Omron CX-Programmer project 新工程 (CX-Programmer 9.72)

# PLC 新PLC1: CP1E E40

## Global symbols (name address type ; comment)
0.00 BOOL  ; 回程1
0.01 BOOL  ; 刹车信号1
0.02 BOOL  ; 系统正常
0.03 BOOL  ; 超程
0.04 BOOL  ; 吹件
0.05 BOOL  ; 刹车信号子2
0.06 BOOL  ; 光电控制1
0.07 BOOL  ; 计数值到
0.08 BOOL  ; 电机启动
0.09 BOOL  ; 电机停止
0.10 BOOL  ; 电机正转
0.11 BOOL  ; 电机反转
100.01 BOOL  ; 运转侦查1
100.02 BOOL  ; 超程指示
100.03 BOOL  ; 凸轮故障
100.04 BOOL  ; 吹件阀
100.05 BOOL  ; 气动泵控制阀
100.06 BOOL  ; 吹件阀2
100.07 BOOL  ; 油泵电机
101.00 BOOL  ; 电机正转
101.01 BOOL  ; 电机反转
101.02 BOOL  ; △运行
101.03 BOOL  ; Y启动
101.04 BOOL  ; 气压指示
101.05 BOOL  ; 连续预置
101.07 BOOL  ; 电机运行
102.00 BOOL  ; 运行侦测2
102.01 BOOL  ; 顶点补正
102.02 BOOL  ; 保护继电器
102.03 BOOL  ; 辅助调整2
102.04 BOOL  ; 润滑故障
102.05 BOOL  ; 双联阀故障指示
102.06 BOOL  ; 异常报警
102.07 BOOL  ; 负荷指示
10.01 BOOL  ; 自动送料阀
13.01 BOOL  ; 电机正反转信号
13.04 BOOL  ; 电机启动信号
14.03 BOOL  ; 运行条件
14.04 BOOL  ; 寸动规范输出
14.05 BOOL  ; 双手同步输出信号
14.06 BOOL  ; 单次信号输出
14.07 BOOL  ; 连续预置信号
14.08 BOOL  ; 误送信号
15.00 BOOL  ; 寸动输出
15.01 BOOL  ; 单次输出
15.03 BOOL  ; 连续输出
15.04 BOOL  ; 调整规范
15.05 BOOL  ; 脚踏输出信号
16.00 BOOL  ; 1秒故障闪烁信号
16.01 BOOL  ; 故障输出
17.00 BOOL  ; 寸动光电遮断信号
18.01 BOOL  ; 功能开关拨动信号
18.03 BOOL  ; 双联阀故障
19.01 BOOL  ; 连续停止信号
19.02 BOOL  ; 连续信号输出
19.05 BOOL  ; 单次运行条件
1.00 BOOL  ; 光电保护
1.01 BOOL  ; 超负荷
1.02 BOOL  ; 脚踏旋钮
1.03 BOOL  ; 双手A
1.04 BOOL  ; 双手B
1.05 BOOL  ; 连续预置
1.06 BOOL  ; 连续停止
1.07 BOOL  ; 急停
1.08 BOOL  ; 气压
1.09 BOOL  ; 送料许可
1.10 BOOL  ; 双联阀故障检测
1.11 BOOL  ; 脚踏开关
200.00 BOOL  ; 润滑屏蔽
200.01 BOOL  ; 气压传感屏蔽
20.02 BOOL  ; 双联阀下降沿
20.03 BOOL  ; 二度落动作
20.04 BOOL  ; 二度落保护
20.05 BOOL  ; 上死点停车
20.06 BOOL  ; 二度落保护
20.07 BOOL  ; 超程保护
22.00 BOOL  ; 单次回程前信号
22.01 BOOL  ; 回程后断回程前
23.00 BOOL  ; 连续信号开始
24.02 BOOL  ; 调整
24.03 BOOL  ; 连续顶点补正信号
24.05 BOOL  ; 反馈不同步
29.00 BOOL  ; 二度落上升沿
29.02 BOOL  ; 超程下降沿
2.00 BOOL  ; 反馈信号1
2.01 BOOL  ; 异常复位
2.02 BOOL  ; 润滑故障检测
2.03 BOOL  ; 寸动信号
2.04 BOOL  ; 单次信号
2.05 BOOL  ; 连续信号
2.06 BOOL  ; 送料接口
2.07 BOOL  ; 误送检知
2.08 BOOL  ; 光电控制2
2.10 BOOL  ; 自动送料
2.11 BOOL  ; 二度落
30.08 BOOL  ; 润滑故障信号
T004 BOOL  ; 双手同步时间
T006 BOOL  ; 连续预置时间
T007 BOOL  ; Y-三角转换时间
T009 BOOL  ; 超负荷信号
T015 BOOL  ; 二度落异常
T018 BOOL  ; 润滑检测开关常通
T019 BOOL  ; 润滑检测开关常闭
T040 BOOL  ; 急停滤波
T042 BOOL  ; 单次双手时间
T045 BOOL  ; 压力处理信号

## Program 新程序1 (cyclic task 0)
Local symbols
p_on BOOL
y20 BOOL

### Section 段1

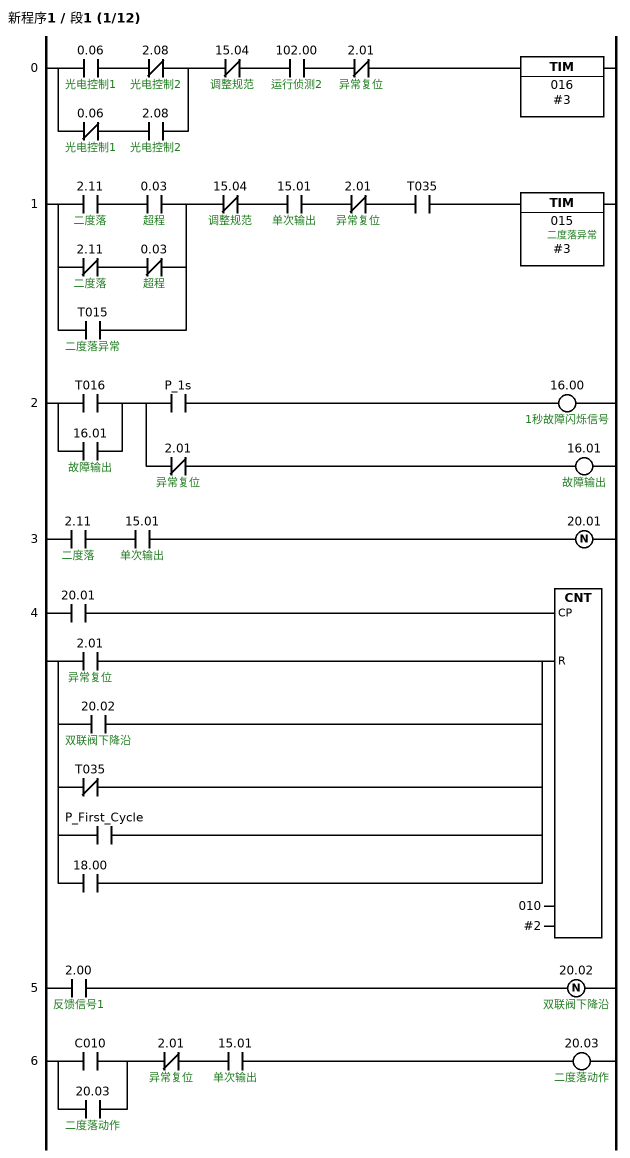
; rung 0
LD 0.06  ; 光电控制1
ANDNOT 2.08  ; 光电控制2
LDNOT 0.06  ; 光电控制1
AND 2.08  ; 光电控制2
ORLD
ANDNOT 15.04  ; 调整规范
AND 102.00  ; 运行侦测2
ANDNOT 2.01  ; 异常复位
TIM 016 #3
; rung 1
LD 2.11  ; 二度落
AND 0.03  ; 超程
LDNOT 2.11  ; 二度落
ANDNOT 0.03  ; 超程
ORLD
OR T015  ; 二度落异常
ANDNOT 15.04  ; 调整规范
AND 15.01  ; 单次输出
ANDNOT 2.01  ; 异常复位
AND T035
TIM 015 #3  ; 二度落异常
; rung 2
LD T016
OR 16.01  ; 故障输出
OUT TR0
AND P_1s
OUT 16.00  ; 1秒故障闪烁信号
LD TR0
ANDNOT 2.01  ; 异常复位
OUT 16.01  ; 故障输出
; rung 3
LD 2.11  ; 二度落
AND 15.01  ; 单次输出
DIFD(014) 20.01
; rung 4
LD 20.01
LD 2.01  ; 异常复位
OR 20.02  ; 双联阀下降沿
ORNOT T035
OR P_First_Cycle
OR 18.00
CNT 010 #2
; rung 5
LD 2.00  ; 反馈信号1
DIFD(014) 20.02  ; 双联阀下降沿
; rung 6
LD C010
OR 20.03  ; 二度落动作
ANDNOT 2.01  ; 异常复位
AND 15.01  ; 单次输出
OUT 20.03  ; 二度落动作

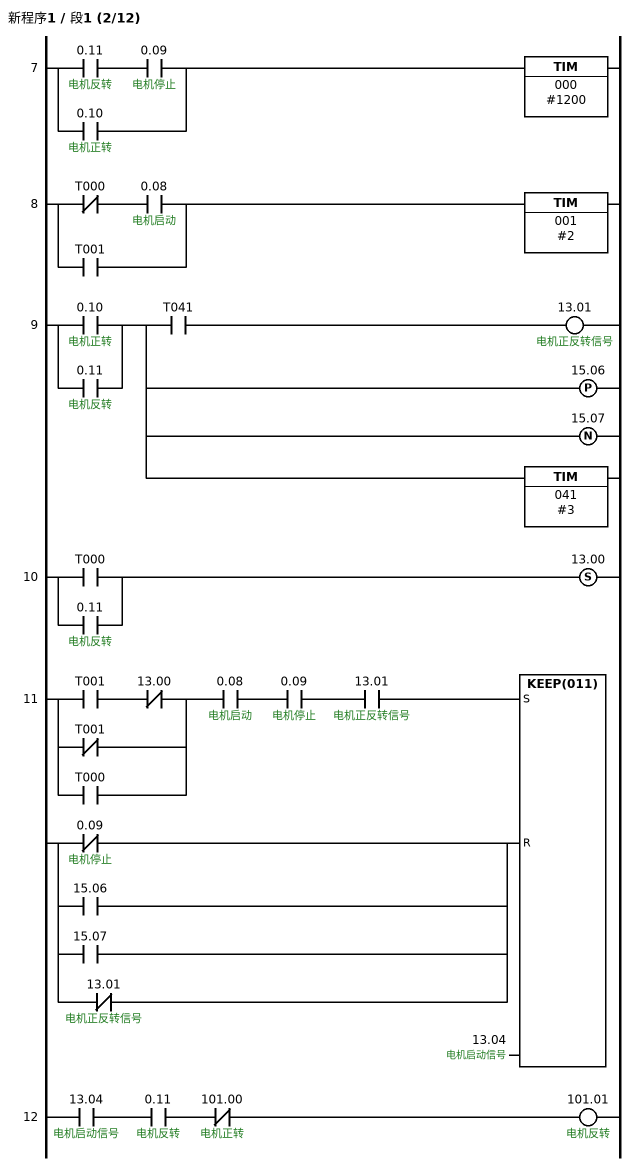
; rung 7
LD 0.11  ; 电机反转
AND 0.09  ; 电机停止
OR 0.10  ; 电机正转
TIM 000 #1200
; rung 8
LDNOT T000
AND 0.08  ; 电机启动
OR T001
TIM 001 #2
; rung 9
LD 0.10  ; 电机正转
OR 0.11  ; 电机反转
OUT TR0
AND T041
OUT 13.01  ; 电机正反转信号
LD TR0
DIFU(013) 15.06
DIFD(014) 15.07
TIM 041 #3
; rung 10
LD T000
OR 0.11  ; 电机反转
SET 13.00
; rung 11
LD T001
ANDNOT 13.00
ORNOT T001
OR T000
AND 0.08  ; 电机启动
AND 0.09  ; 电机停止
AND 13.01  ; 电机正反转信号
LDNOT 0.09  ; 电机停止
OR 15.06
OR 15.07
ORNOT 13.01  ; 电机正反转信号
KEEP(011) 13.04  ; 电机启动信号
; rung 12
LD 13.04  ; 电机启动信号
AND 0.11  ; 电机反转
ANDNOT 101.00  ; 电机正转
OUT 101.01  ; 电机反转

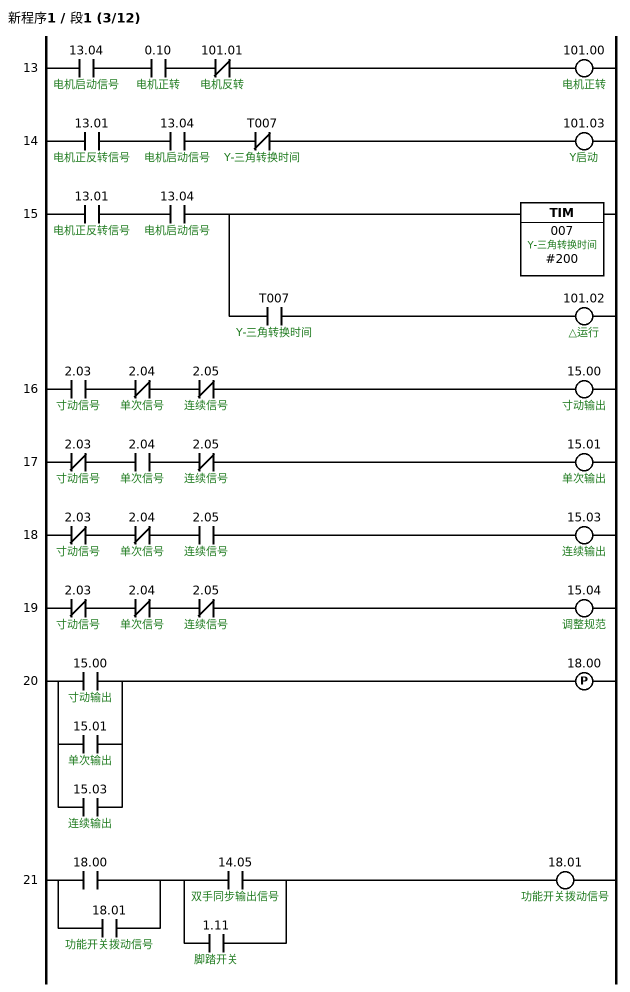
; rung 13
LD 13.04  ; 电机启动信号
AND 0.10  ; 电机正转
ANDNOT 101.01  ; 电机反转
OUT 101.00  ; 电机正转
; rung 14
LD 13.01  ; 电机正反转信号
AND 13.04  ; 电机启动信号
ANDNOT T007  ; Y-三角转换时间
OUT 101.03  ; Y启动
; rung 15
LD 13.01  ; 电机正反转信号
AND 13.04  ; 电机启动信号
TIM 007 #200  ; Y-三角转换时间
AND T007  ; Y-三角转换时间
OUT 101.02  ; △运行
; rung 16
LD 2.03  ; 寸动信号
ANDNOT 2.04  ; 单次信号
ANDNOT 2.05  ; 连续信号
OUT 15.00  ; 寸动输出
; rung 17
LDNOT 2.03  ; 寸动信号
AND 2.04  ; 单次信号
ANDNOT 2.05  ; 连续信号
OUT 15.01  ; 单次输出
; rung 18
LDNOT 2.03  ; 寸动信号
ANDNOT 2.04  ; 单次信号
AND 2.05  ; 连续信号
OUT 15.03  ; 连续输出
; rung 19
LDNOT 2.03  ; 寸动信号
ANDNOT 2.04  ; 单次信号
ANDNOT 2.05  ; 连续信号
OUT 15.04  ; 调整规范
; rung 20
LD 15.00  ; 寸动输出
OR 15.01  ; 单次输出
OR 15.03  ; 连续输出
DIFU(013) 18.00
; rung 21
LD 18.00
OR 18.01  ; 功能开关拨动信号
LD 14.05  ; 双手同步输出信号
OR 1.11  ; 脚踏开关
ANDLD
OUT 18.01  ; 功能开关拨动信号

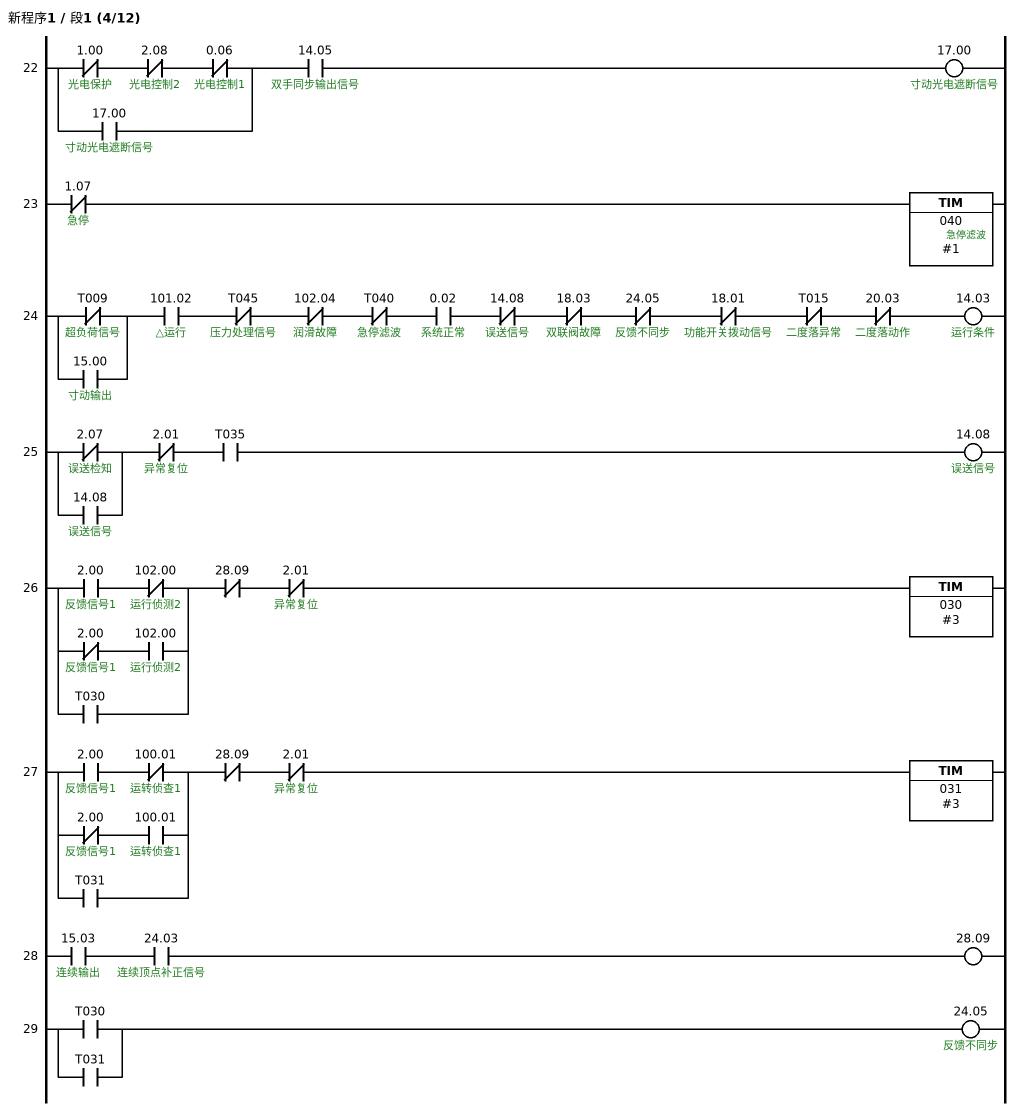
; rung 22
LDNOT 1.00  ; 光电保护
ANDNOT 2.08  ; 光电控制2
ANDNOT 0.06  ; 光电控制1
OR 17.00  ; 寸动光电遮断信号
AND 14.05  ; 双手同步输出信号
OUT 17.00  ; 寸动光电遮断信号
; rung 23
LDNOT 1.07  ; 急停
TIM 040 #1  ; 急停滤波
; rung 24
LDNOT T009  ; 超负荷信号
OR 15.00  ; 寸动输出
AND 101.02  ; △运行
ANDNOT T045  ; 压力处理信号
ANDNOT 102.04  ; 润滑故障
ANDNOT T040  ; 急停滤波
AND 0.02  ; 系统正常
ANDNOT 14.08  ; 误送信号
ANDNOT 18.03  ; 双联阀故障
ANDNOT 24.05  ; 反馈不同步
ANDNOT 18.01  ; 功能开关拨动信号
ANDNOT T015  ; 二度落异常
ANDNOT 20.03  ; 二度落动作
OUT 14.03  ; 运行条件
; rung 25
LDNOT 2.07  ; 误送检知
OR 14.08  ; 误送信号
ANDNOT 2.01  ; 异常复位
AND T035
OUT 14.08  ; 误送信号
; rung 26
LD 2.00  ; 反馈信号1
ANDNOT 102.00  ; 运行侦测2
LDNOT 2.00  ; 反馈信号1
AND 102.00  ; 运行侦测2
ORLD
OR T030
ANDNOT 28.09
ANDNOT 2.01  ; 异常复位
TIM 030 #3
; rung 27
LD 2.00  ; 反馈信号1
ANDNOT 100.01  ; 运转侦查1
LDNOT 2.00  ; 反馈信号1
AND 100.01  ; 运转侦查1
ORLD
OR T031
ANDNOT 28.09
ANDNOT 2.01  ; 异常复位
TIM 031 #3
; rung 28
LD 15.03  ; 连续输出
AND 24.03  ; 连续顶点补正信号
OUT 28.09
; rung 29
LD T030
OR T031
OUT 24.05  ; 反馈不同步

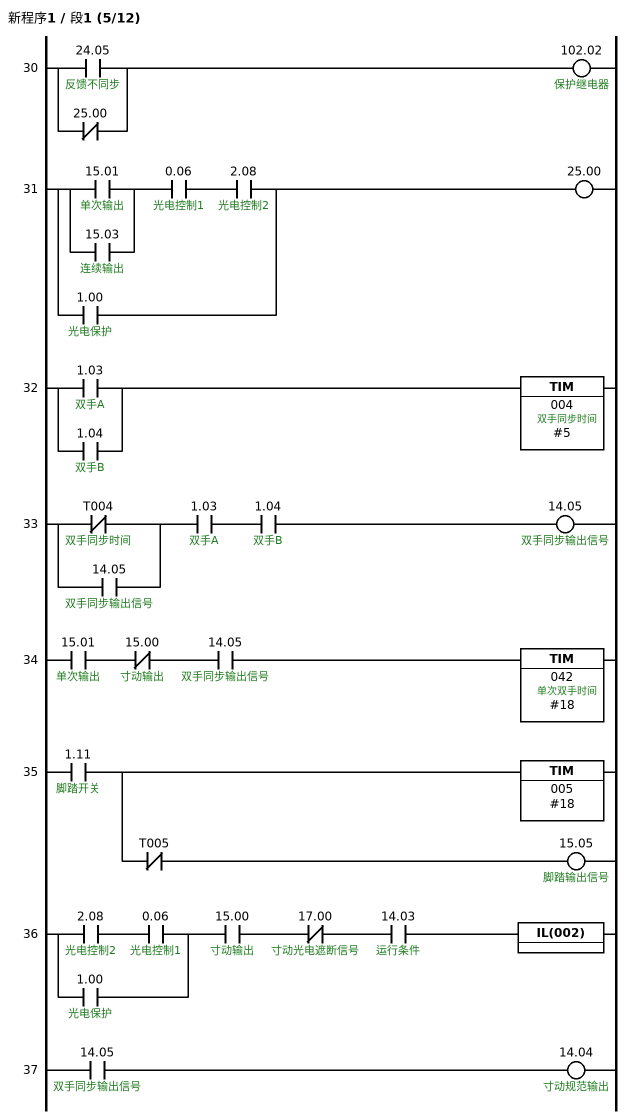
; rung 30
LD 24.05  ; 反馈不同步
ORNOT 25.00
OUT 102.02  ; 保护继电器
; rung 31
LD 15.01  ; 单次输出
OR 15.03  ; 连续输出
AND 0.06  ; 光电控制1
AND 2.08  ; 光电控制2
OR 1.00  ; 光电保护
OUT 25.00
; rung 32
LD 1.03  ; 双手A
OR 1.04  ; 双手B
TIM 004 #5  ; 双手同步时间
; rung 33
LDNOT T004  ; 双手同步时间
OR 14.05  ; 双手同步输出信号
AND 1.03  ; 双手A
AND 1.04  ; 双手B
OUT 14.05  ; 双手同步输出信号
; rung 34
LD 15.01  ; 单次输出
ANDNOT 15.00  ; 寸动输出
AND 14.05  ; 双手同步输出信号
TIM 042 #18  ; 单次双手时间
; rung 35
LD 1.11  ; 脚踏开关
TIM 005 #18
ANDNOT T005
OUT 15.05  ; 脚踏输出信号
; rung 36
LD 2.08  ; 光电控制2
AND 0.06  ; 光电控制1
OR 1.00  ; 光电保护
AND 15.00  ; 寸动输出
ANDNOT 17.00  ; 寸动光电遮断信号
AND 14.03  ; 运行条件
IL(002)
; rung 37
LD 14.05  ; 双手同步输出信号
OUT 14.04  ; 寸动规范输出

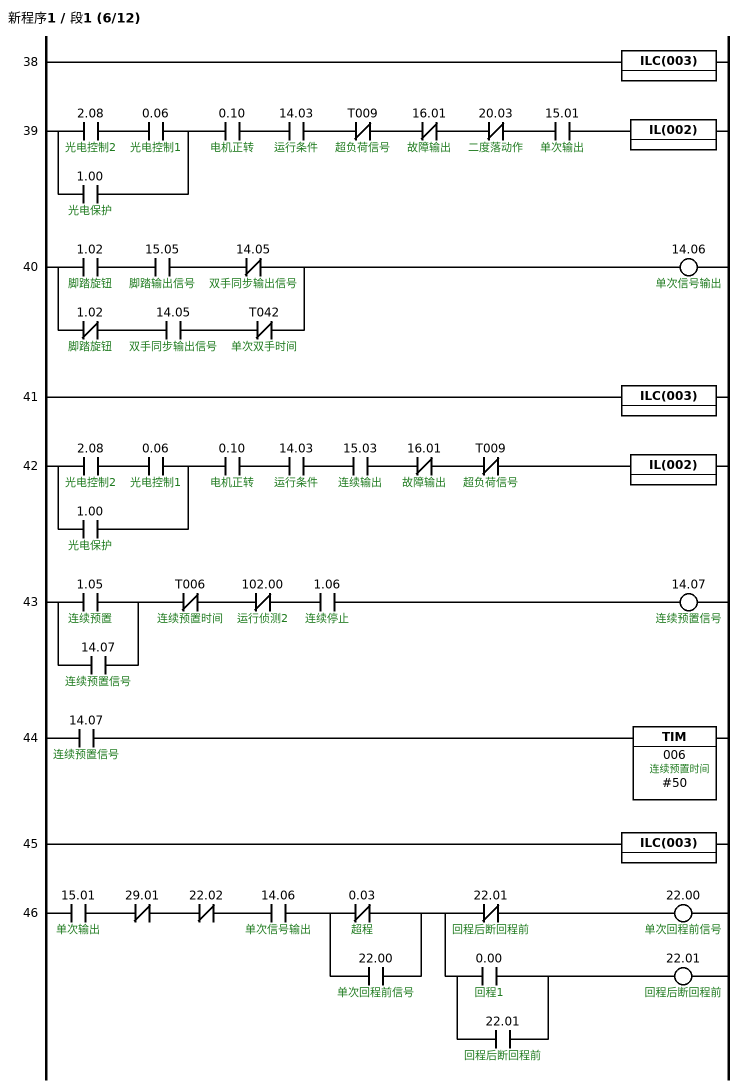
; rung 38
ILC(003)
; rung 39
LD 2.08  ; 光电控制2
AND 0.06  ; 光电控制1
OR 1.00  ; 光电保护
AND 0.10  ; 电机正转
AND 14.03  ; 运行条件
ANDNOT T009  ; 超负荷信号
ANDNOT 16.01  ; 故障输出
ANDNOT 20.03  ; 二度落动作
AND 15.01  ; 单次输出
IL(002)
; rung 40
LD 1.02  ; 脚踏旋钮
AND 15.05  ; 脚踏输出信号
ANDNOT 14.05  ; 双手同步输出信号
LDNOT 1.02  ; 脚踏旋钮
AND 14.05  ; 双手同步输出信号
ANDNOT T042  ; 单次双手时间
ORLD
OUT 14.06  ; 单次信号输出
; rung 41
ILC(003)
; rung 42
LD 2.08  ; 光电控制2
AND 0.06  ; 光电控制1
OR 1.00  ; 光电保护
AND 0.10  ; 电机正转
AND 14.03  ; 运行条件
AND 15.03  ; 连续输出
ANDNOT 16.01  ; 故障输出
ANDNOT T009  ; 超负荷信号
IL(002)
; rung 43
LD 1.05  ; 连续预置
OR 14.07  ; 连续预置信号
ANDNOT T006  ; 连续预置时间
ANDNOT 102.00  ; 运行侦测2
AND 1.06  ; 连续停止
OUT 14.07  ; 连续预置信号
; rung 44
LD 14.07  ; 连续预置信号
TIM 006 #50  ; 连续预置时间
; rung 45
ILC(003)
; rung 46
LD 15.01  ; 单次输出
ANDNOT 29.01
ANDNOT 22.02
AND 14.06  ; 单次信号输出
LDNOT 0.03  ; 超程
OR 22.00  ; 单次回程前信号
ANDLD
OUT TR0
ANDNOT 22.01  ; 回程后断回程前
OUT 22.00  ; 单次回程前信号
LD TR0
LD 0.00  ; 回程1
OR 22.01  ; 回程后断回程前
ANDLD
OUT 22.01  ; 回程后断回程前

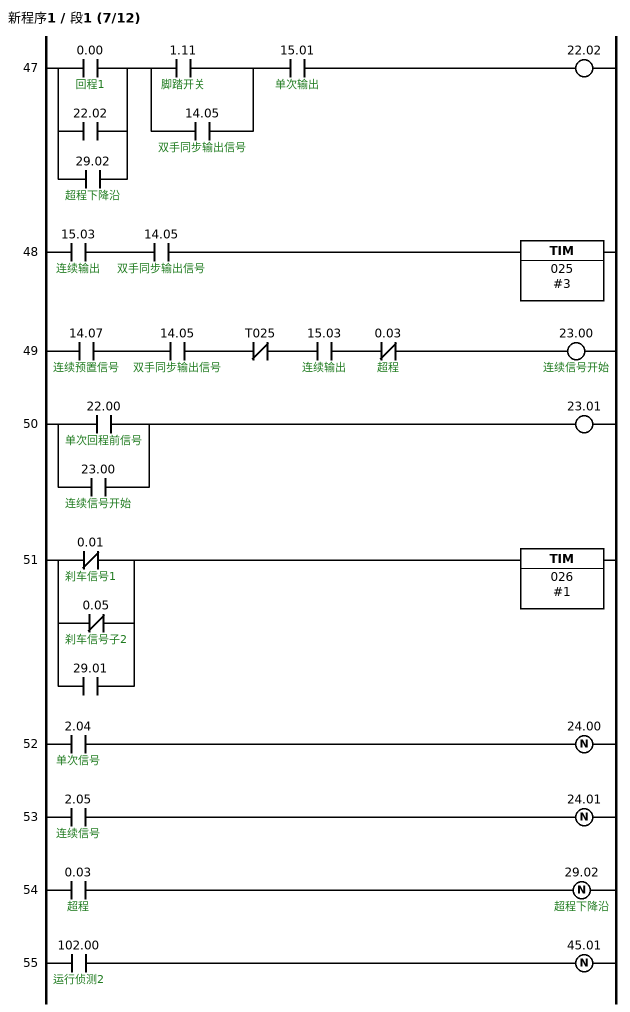
; rung 47
LD 0.00  ; 回程1
OR 22.02
OR 29.02  ; 超程下降沿
LD 1.11  ; 脚踏开关
OR 14.05  ; 双手同步输出信号
ANDLD
AND 15.01  ; 单次输出
OUT 22.02
; rung 48
LD 15.03  ; 连续输出
AND 14.05  ; 双手同步输出信号
TIM 025 #3
; rung 49
LD 14.07  ; 连续预置信号
AND 14.05  ; 双手同步输出信号
ANDNOT T025
AND 15.03  ; 连续输出
ANDNOT 0.03  ; 超程
OUT 23.00  ; 连续信号开始
; rung 50
LD 22.00  ; 单次回程前信号
OR 23.00  ; 连续信号开始
OUT 23.01
; rung 51
LDNOT 0.01  ; 刹车信号1
ORNOT 0.05  ; 刹车信号子2
OR 29.01
TIM 026 #1
; rung 52
LD 2.04  ; 单次信号
DIFD(014) 24.00
; rung 53
LD 2.05  ; 连续信号
DIFD(014) 24.01
; rung 54
LD 0.03  ; 超程
DIFD(014) 29.02  ; 超程下降沿
; rung 55
LD 102.00  ; 运行侦测2
DIFD(014) 45.01

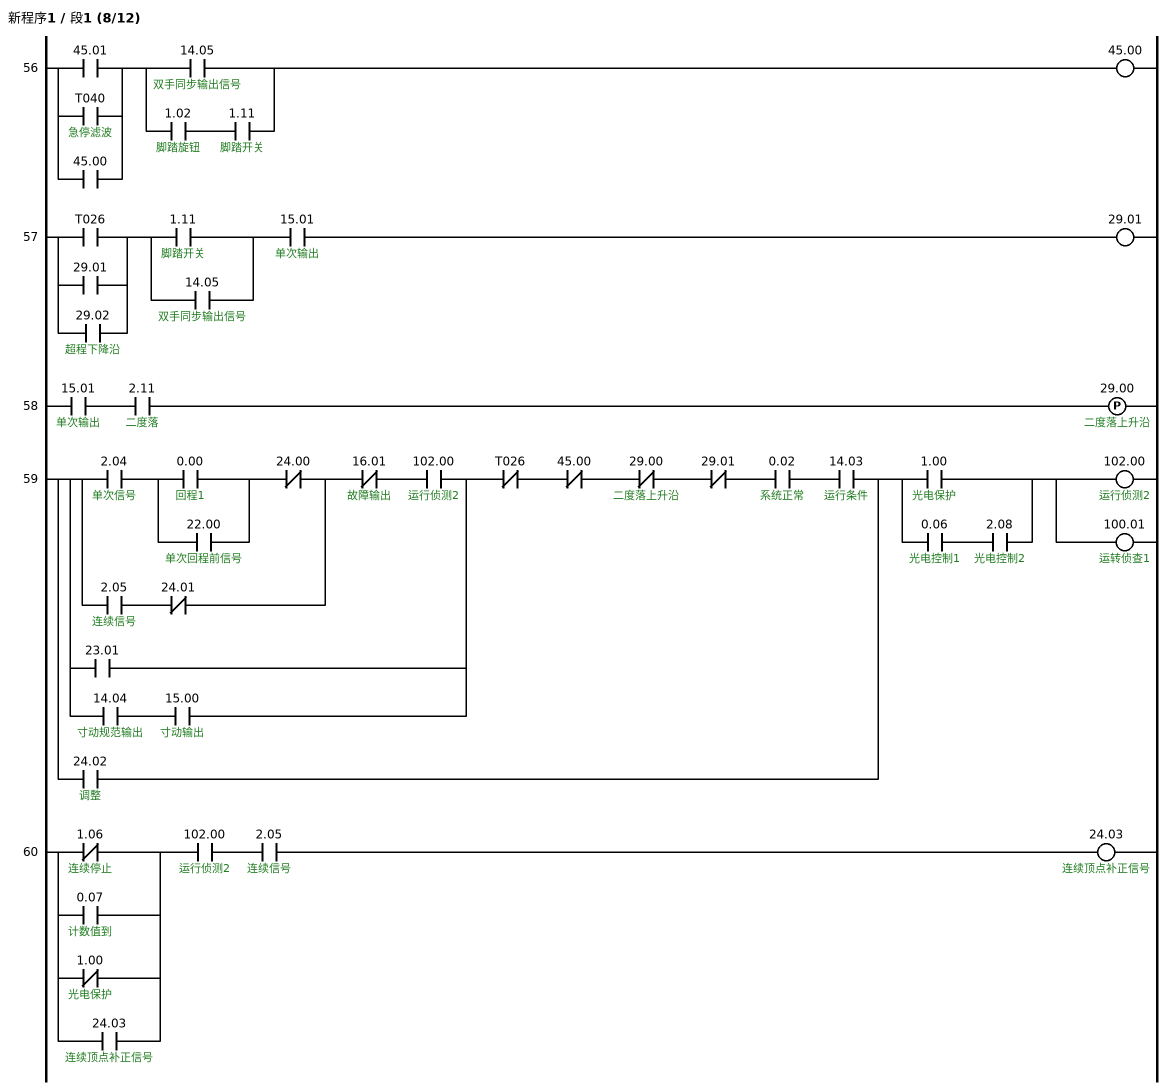
; rung 56
LD 45.01
OR T040  ; 急停滤波
OR 45.00
LD 14.05  ; 双手同步输出信号
LD 1.02  ; 脚踏旋钮
AND 1.11  ; 脚踏开关
ORLD
ANDLD
OUT 45.00
; rung 57
LD T026
OR 29.01
OR 29.02  ; 超程下降沿
LD 1.11  ; 脚踏开关
OR 14.05  ; 双手同步输出信号
ANDLD
AND 15.01  ; 单次输出
OUT 29.01
; rung 58
LD 15.01  ; 单次输出
AND 2.11  ; 二度落
DIFU(013) 29.00  ; 二度落上升沿
; rung 59
LD 2.04  ; 单次信号
LD 0.00  ; 回程1
OR 22.00  ; 单次回程前信号
ANDLD
ANDNOT 24.00
LD 2.05  ; 连续信号
ANDNOT 24.01
ORLD
ANDNOT 16.01  ; 故障输出
AND 102.00  ; 运行侦测2
OR 23.01
LD 14.04  ; 寸动规范输出
AND 15.00  ; 寸动输出
ORLD
ANDNOT T026
ANDNOT 45.00
ANDNOT 29.00  ; 二度落上升沿
ANDNOT 29.01
AND 0.02  ; 系统正常
AND 14.03  ; 运行条件
OR 24.02  ; 调整
LD 1.00  ; 光电保护
LD 0.06  ; 光电控制1
AND 2.08  ; 光电控制2
ORLD
ANDLD
OUT 102.00  ; 运行侦测2
OUT 100.01  ; 运转侦查1
; rung 60
LDNOT 1.06  ; 连续停止
OR 0.07  ; 计数值到
ORNOT 1.00  ; 光电保护
OR 24.03  ; 连续顶点补正信号
AND 102.00  ; 运行侦测2
AND 2.05  ; 连续信号
OUT 24.03  ; 连续顶点补正信号

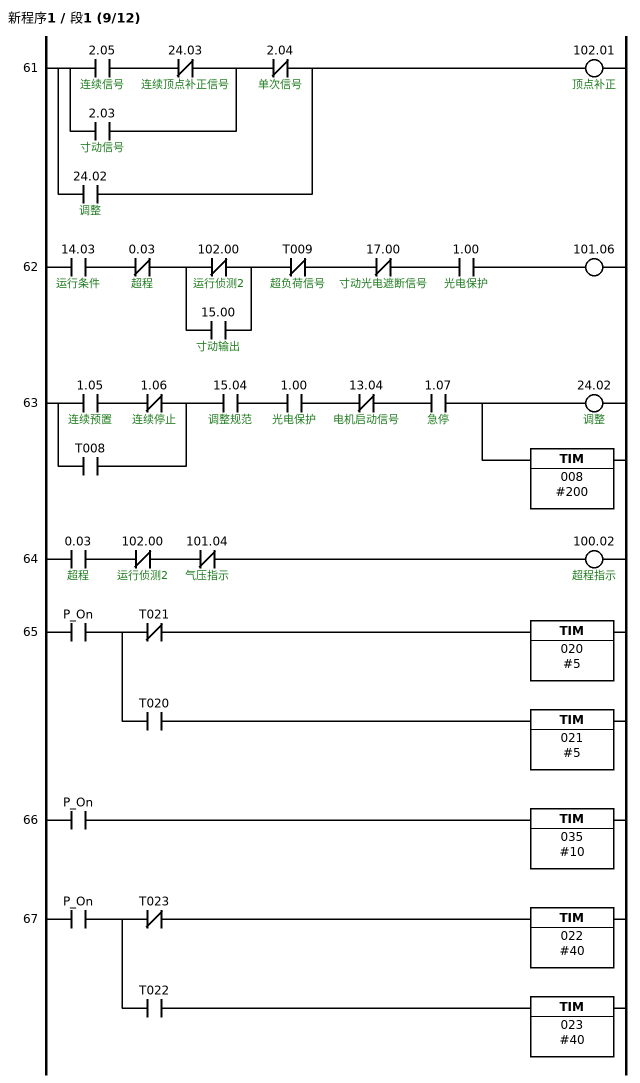
; rung 61
LD 2.05  ; 连续信号
ANDNOT 24.03  ; 连续顶点补正信号
OR 2.03  ; 寸动信号
ANDNOT 2.04  ; 单次信号
OR 24.02  ; 调整
OUT 102.01  ; 顶点补正
; rung 62
LD 14.03  ; 运行条件
ANDNOT 0.03  ; 超程
LDNOT 102.00  ; 运行侦测2
OR 15.00  ; 寸动输出
ANDLD
ANDNOT T009  ; 超负荷信号
ANDNOT 17.00  ; 寸动光电遮断信号
AND 1.00  ; 光电保护
OUT 101.06
; rung 63
LD 1.05  ; 连续预置
ANDNOT 1.06  ; 连续停止
OR T008
AND 15.04  ; 调整规范
AND 1.00  ; 光电保护
ANDNOT 13.04  ; 电机启动信号
AND 1.07  ; 急停
OUT 24.02  ; 调整
TIM 008 #200
; rung 64
LD 0.03  ; 超程
ANDNOT 102.00  ; 运行侦测2
ANDNOT 101.04  ; 气压指示
OUT 100.02  ; 超程指示
; rung 65
LD P_On
OUT TR0
ANDNOT T021
TIM 020 #5
LD TR0
AND T020
TIM 021 #5
; rung 66
LD P_On
TIM 035 #10
; rung 67
LD P_On
OUT TR0
ANDNOT T023
TIM 022 #40
LD TR0
AND T022
TIM 023 #40

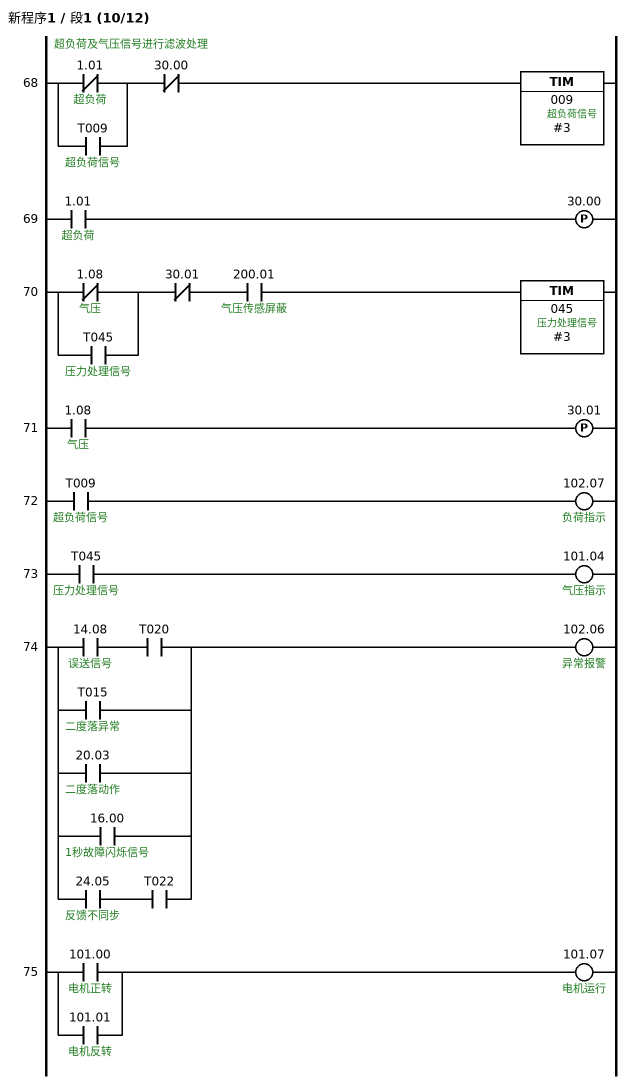
; rung 68: 超负荷及气压信号进行滤波处理
LDNOT 1.01  ; 超负荷
OR T009  ; 超负荷信号
ANDNOT 30.00
TIM 009 #3  ; 超负荷信号
; rung 69
LD 1.01  ; 超负荷
DIFU(013) 30.00
; rung 70
LDNOT 1.08  ; 气压
OR T045  ; 压力处理信号
ANDNOT 30.01
AND 200.01  ; 气压传感屏蔽
TIM 045 #3  ; 压力处理信号
; rung 71
LD 1.08  ; 气压
DIFU(013) 30.01
; rung 72
LD T009  ; 超负荷信号
OUT 102.07  ; 负荷指示
; rung 73
LD T045  ; 压力处理信号
OUT 101.04  ; 气压指示
; rung 74
LD 14.08  ; 误送信号
AND T020
OR T015  ; 二度落异常
OR 20.03  ; 二度落动作
OR 16.00  ; 1秒故障闪烁信号
LD 24.05  ; 反馈不同步
AND T022
ORLD
OUT 102.06  ; 异常报警
; rung 75
LD 101.00  ; 电机正转
OR 101.01  ; 电机反转
OUT 101.07  ; 电机运行

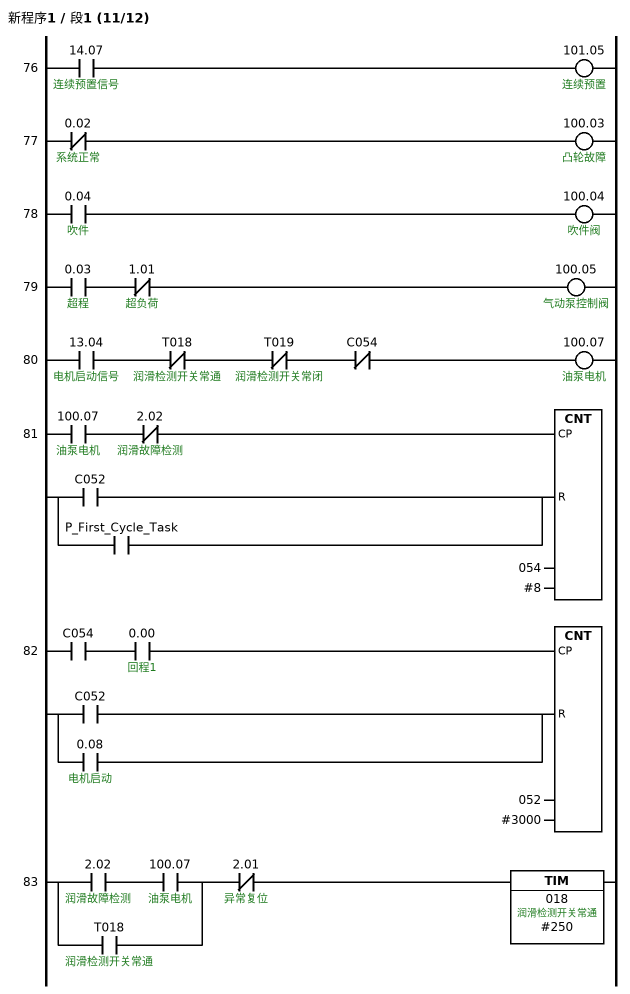
; rung 76
LD 14.07  ; 连续预置信号
OUT 101.05  ; 连续预置
; rung 77
LDNOT 0.02  ; 系统正常
OUT 100.03  ; 凸轮故障
; rung 78
LD 0.04  ; 吹件
OUT 100.04  ; 吹件阀
; rung 79
LD 0.03  ; 超程
ANDNOT 1.01  ; 超负荷
OUT 100.05  ; 气动泵控制阀
; rung 80
LD 13.04  ; 电机启动信号
ANDNOT T018  ; 润滑检测开关常通
ANDNOT T019  ; 润滑检测开关常闭
ANDNOT C054
OUT 100.07  ; 油泵电机
; rung 81
LD 100.07  ; 油泵电机
ANDNOT 2.02  ; 润滑故障检测
LD C052
OR P_First_Cycle_Task
CNT 054 #8
; rung 82
LD C054
AND 0.00  ; 回程1
LD C052
OR 0.08  ; 电机启动
CNT 052 #3000
; rung 83
LD 2.02  ; 润滑故障检测
AND 100.07  ; 油泵电机
OR T018  ; 润滑检测开关常通
ANDNOT 2.01  ; 异常复位
TIM 018 #250  ; 润滑检测开关常通

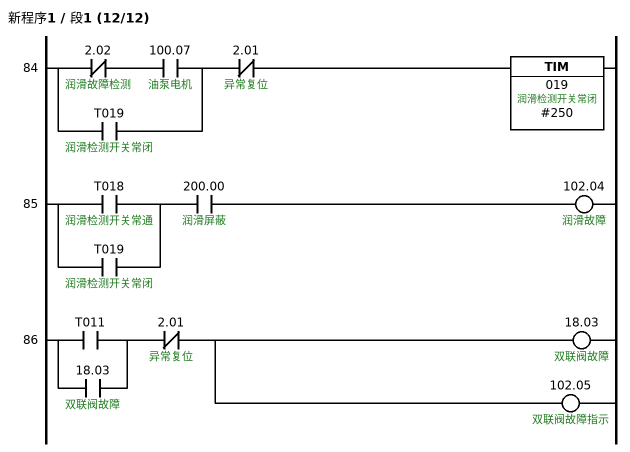
; rung 84
LDNOT 2.02  ; 润滑故障检测
AND 100.07  ; 油泵电机
OR T019  ; 润滑检测开关常闭
ANDNOT 2.01  ; 异常复位
TIM 019 #250  ; 润滑检测开关常闭
; rung 85
LD T018  ; 润滑检测开关常通
OR T019  ; 润滑检测开关常闭
AND 200.00  ; 润滑屏蔽
OUT 102.04  ; 润滑故障
; rung 86
LD T011
OR 18.03  ; 双联阀故障
ANDNOT 2.01  ; 异常复位
OUT 18.03  ; 双联阀故障
OUT 102.05  ; 双联阀故障指示
; rung 87
END(001)